% RSLogix 500 project Schwebekörper-Durchflussmesser.RSS, saved by version 8.30.00.16 %
PROJECT "UNTITLED"    % processor: Bul.1763 MicroLogix 1100 Series B %

PROGRAM FILES
  LAD 2   8 rungs

DATA FILES
  O0 OUTPUT  4 elements
  I1 INPUT  6 elements
  S2 STATUS  66 elements
  B3 BINARY  1 elements
  T4 TIMER  2 elements
  C5 COUNTER  1 elements
  R6 CONTROL  1 elements
  N7 INTEGER  2 elements
  F8 FLOAT  3 elements

LADDER 2
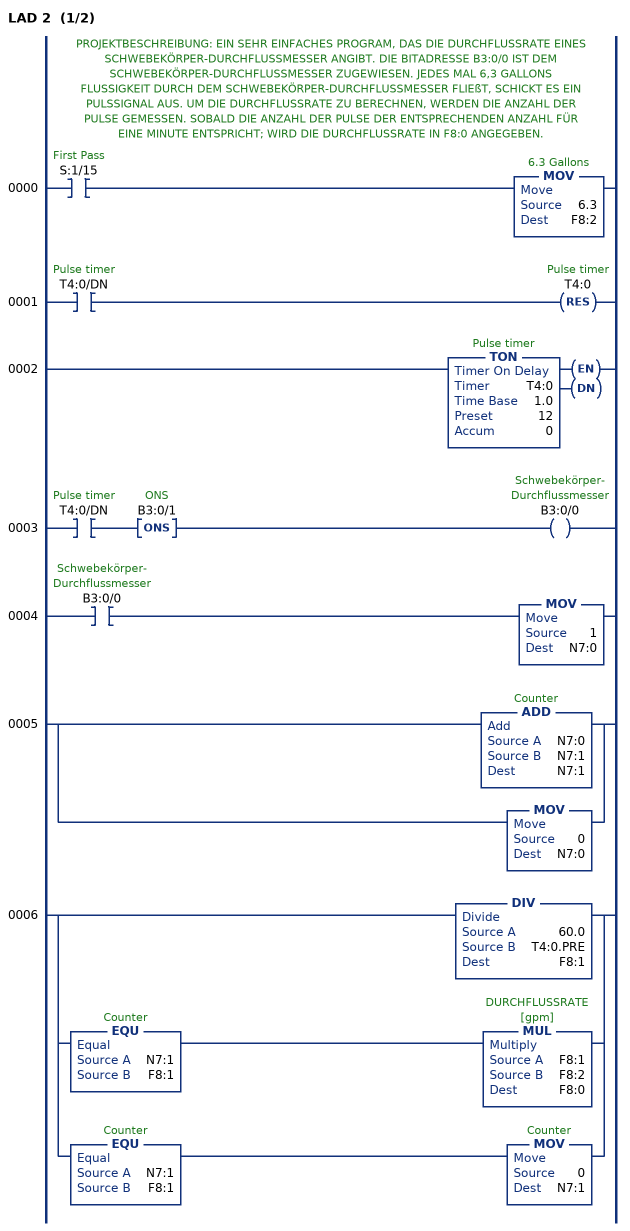
% Rung: 0 %
% PROJEKTBESCHREIBUNG: EIN SEHR EINFACHES PROGRAM, DAS DIE DURCHFLUSSRATE EINES SCHWEBEKÖRPER-DURCHFLUSSMESSER ANGIBT. DIE BITADRESSE B3:0/0 IST DEM SCHWEBEKÖRPER-DURCHFLUSSMESSER ZUGEWIESEN. JEDES MAL 6,3 GALLONS FLUSSIGKEIT DURCH DEM SCHWEBEKÖRPER-DURCHFLUSSMESSER FLIEßT, SCHICKT ES EIN PULSSIGNAL AUS. UM DIE DURCHFLUSSRATE ZU BERECHNEN, WERDEN DIE ANZAHL DER PULSE GEMESSEN. SOBALD DIE ANZAHL DER PULSE DER ENTSPRECHENDEN ANZAHL FÜR EINE MINUTE ENTSPRICHT; WIRD DIE DURCHFLUSSRATE IN F8:0 ANGEGEBEN. %
SOR XIC S:1/15 MOV 6.3 F8:2 EOR
%   S:1/15  "First Pass" %
%   F8:2  "6.3 Gallons" %
% Rung: 1 %
SOR XIC T4:0/DN RES T4:0 EOR
%   T4:0  "Pulse timer" %
% Rung: 2 %
SOR TON T4:0 1.0 12 0 EOR
%   T4:0  "Pulse timer" %
% Rung: 3 %
SOR XIC T4:0/DN ONS B3:0/1 OTE B3:0/0 EOR
%   T4:0  "Pulse timer" %
%   B3:0/1  "ONS" %
%   B3:0/0  "Schwebekörper- Durchflussmesser" %
% Rung: 4 %
SOR XIC B3:0/0 MOV 1 N7:0 EOR
%   B3:0/0  "Schwebekörper- Durchflussmesser" %
% Rung: 5 %
SOR BST ADD N7:0 N7:1 N7:1 NXB MOV 0 N7:0 BND EOR
%   N7:1  "Counter" %
% Rung: 6 %
SOR BST DIV 60.0 T4:0.PRE F8:1 NXB EQU N7:1 F8:1 MUL F8:1 F8:2 F8:0 NXB EQU N7:1 F8:1 MOV 0 N7:1 BND EOR
%   T4:0  "Pulse timer" %
%   N7:1  "Counter" %
%   F8:2  "6.3 Gallons" %
%   F8:0  "DURCHFLUSSRATE [gpm]" %

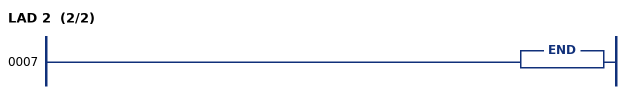
% Rung: 7 %
SOR END EOR

OTHER DOCUMENTED ADDRESSES
  T4:1  "Counting Pulses"

DATA TABLE (non-zero values as saved)
DATA T4
% .PRE .ACC %
% T4:0 % 12 0
